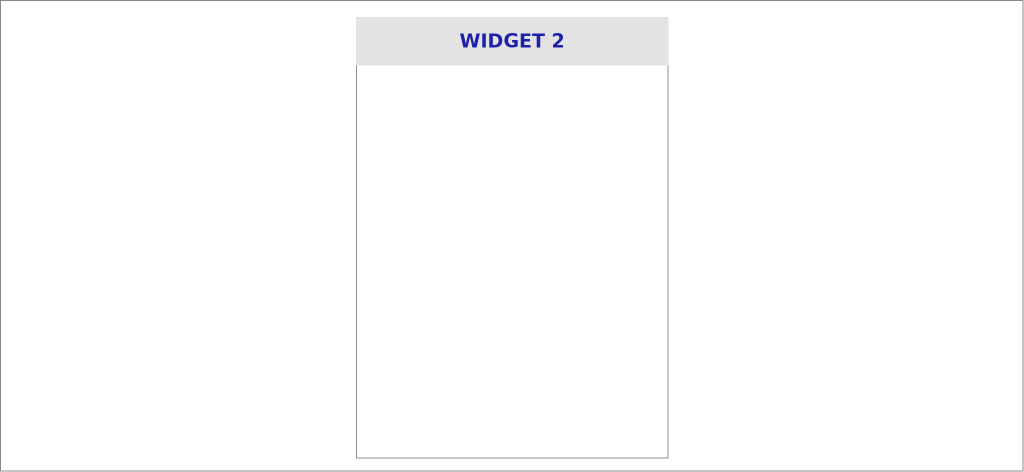
VISUALIZATION _002_Blank_2  // 1024x472
    GroupBox (356,16 312x442)
        Rectangle (0,1 312x48), "WIDGET 2"
END_VISUALIZATION

(* stored: Version 1.1.0.1, ProductVersion 3.1.4022.18
   Visu _002_Blank_2: Id {82a5e455-7bbf-4d55-a010-ee527d0a0c02} *)
